FUNCTION_BLOCK AQ_MERGE_8 (* Fan-In: Merges 8 AQ into 1 AQ adapter *)
  (* Standard: 61499-2; Description: Copyright (c) 2026 Meisterschulen am Ostbahnhof SPDX-License-Identifier: EPL-2.0 *)
  (* Version 1.0, 2026-05-16, Franz Höpfinger, Meisterschulen am Ostbahnhof, Initial Version *)
  PACKAGE adapter::events::unidirectional;
  IMPORT eclipse4diac::core::GenericClassName;
  {SET_ATTRIBUTE(eclipse4diac::core::GenericClassName, 'GEN_AQ_MERGE')}
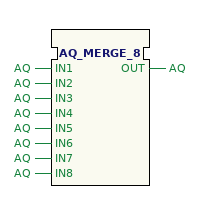
  SOCKETS
    IN1 : adapter::types::unidirectional::AQ;
    IN2 : adapter::types::unidirectional::AQ;
    IN3 : adapter::types::unidirectional::AQ;
    IN4 : adapter::types::unidirectional::AQ;
    IN5 : adapter::types::unidirectional::AQ;
    IN6 : adapter::types::unidirectional::AQ;
    IN7 : adapter::types::unidirectional::AQ;
    IN8 : adapter::types::unidirectional::AQ;
  END_SOCKETS
  PLUGS
    OUT : adapter::types::unidirectional::AQ;
  END_PLUGS
END_FUNCTION_BLOCK
